FUNCTION_BLOCK Multicast_TwoCTL (* Composite Function Block Type *)
  (* Standard: 61499-2 *)
  (* Version 0.2, 2003-12-05, JHC, Rockwell Automation, Renamed from NEWCOMPFB. *)
  (* Version 0.1, 2002-01-08, JHC, Rockwell Automation, Added DLY FB as example. *)
  (* Version 0.0, 2000-05-27, JHC, Rockwell Automation *)
  (* Compiler header: package fb.rt.cs725; *)
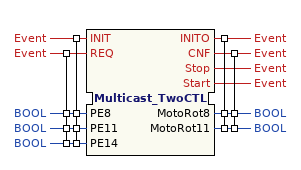
  EVENT_INPUT
    INIT WITH PE8, PE11, PE14; (* Initialization Request *)
    REQ WITH PE8, PE14, PE11; (* Normal Execution Request *)
  END_EVENT
  EVENT_OUTPUT
    INITO WITH MotoRot8, MotoRot11; (* Initialization Confirm *)
    CNF WITH MotoRot8, MotoRot11; (* Execution Confirmation *)
    Stop;
    Start;
  END_EVENT
  VAR_INPUT
    PE8 : BOOL; (* Input event qualifier *)
    PE11 : BOOL;
    PE14 : BOOL;
  END_VAR
  VAR_OUTPUT
    MotoRot8 : BOOL; (* Output event qualifier *)
    MotoRot11 : BOOL;
  END_VAR
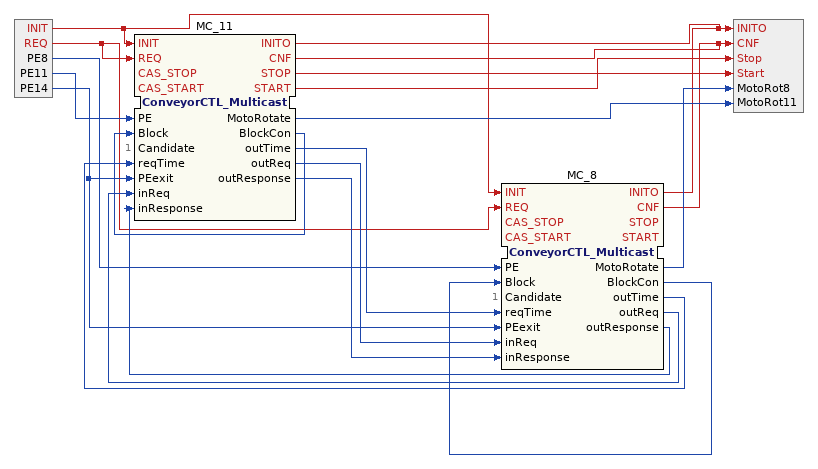
  FBS
    MC_8 : ConveyorCTL_Multicast(Candidate := 1);
    MC_11 : ConveyorCTL_Multicast(Candidate := 1);
  END_FBS
  EVENT_CONNECTIONS
    MC_11.STOP TO Stop;
    MC_11.START TO Start;
    MC_8.INITO TO INITO;
    MC_8.CNF TO CNF;
    REQ TO MC_8.REQ;
    REQ TO MC_11.REQ;
    INIT TO MC_11.INIT;
    INIT TO MC_8.INIT;
    MC_11.INITO TO INITO;
    MC_11.CNF TO CNF;
  END_CONNECTIONS
  DATA_CONNECTIONS
    PE11 TO MC_11.PE;
    PE8 TO MC_8.PE;
    PE14 TO MC_11.PEexit;
    PE14 TO MC_8.PEexit;
    MC_11.MotoRotate TO MotoRot11;
    MC_8.MotoRotate TO MotoRot8;
    MC_8.BlockCon TO MC_8.Block;
    MC_11.BlockCon TO MC_11.Block;
    MC_8.outReq TO MC_11.inReq;
    MC_8.outResponse TO MC_11.inResponse;
    MC_8.outTime TO MC_11.reqTime;
    MC_11.outTime TO MC_8.reqTime;
    MC_11.outReq TO MC_8.inReq;
    MC_11.outResponse TO MC_8.inResponse;
  END_CONNECTIONS
END_FUNCTION_BLOCK
